DATA_BLOCK "DB %%TAG%%"
{ S7_Optimized_Access := 'FALSE' }
VERSION : 0.1
NON_RETAIN
"@pc FB500 monAI _New"

BEGIN
   SAMPLE_T := 0.1;
   HMI_SIM := TRUE;
   "enAlm AH" := TRUE;
   "enAlm WH" := TRUE;
   "enAlm WL" := TRUE;
   "enAlm AL" := TRUE;
   "enAlm CSF" := TRUE;
   "enAction AH" := TRUE;
   "enAction WH" := TRUE;
   "enAction WL" := TRUE;
   "enAction AL" := TRUE;
   "enAction CSF" := TRUE;
   "exist AH" := FALSE;
   "exist WH" := FALSE;
   "exist WL" := FALSE;
   "exist AL" := FALSE;
   "exist CSF" := FALSE;
   "enCalc AH" := TRUE;
   "enCalc WH" := TRUE;
   "enCalc WL" := TRUE;
   "enCalc AL" := TRUE;
   "enCalc CSF" := TRUE;
   hmiContrBYP := FALSE;
   AH_isTRIP := TRUE;
   WH_isTRIP := FALSE;
   WL_isTRIP := FALSE;
   AL_isTRIP := TRUE;
   CSF_isTRIP := TRUE;
   enSUBS := FALSE;
   pvSUBS := 0.0;
   inDIR := FALSE;
   pvDIR := 0.0;
   inDIR_upLim := 400.0;
   inDIR_loLim := -200.0;
   inChannel := 0;
   inCARD_upLim := 20.0;
   inCARD_loLim := 4.0;
   inRAW_upLim := 27648.0;
   inRAW_loLim := 0.0;
   NM_upLim := 400.0;
   NM_loLim := -200.0;
   CSF_External := FALSE;
   CSF_UpLim := 30000.0;
   CSF_loLim := -30000.0;
   HYS := 0.0;
   timSET_AHOn := 0.0;
   timSET_AHOff := 2.0;
   timSET_WHOn := 0.0;
   timSET_WHOff := 2.0;
   timSET_WLOn := 0.0;
   timSET_WLOff := 2.0;
   timSET_ALOn := 0.0;
   timSET_ALOff := 2.0;
   timSET_CSFOn := 0.0;
   timSET_CSFOff := 2.0;
   qPV := 0.0;
   qmeasPV := 0.0;
   qCARD := 0.0;
   "qAlm AH" := FALSE;
   "qAlm WH" := FALSE;
   "qAlm WL" := FALSE;
   "qAlm AL" := FALSE;
   "qAlm CSF" := FALSE;
   "qAction AH" := FALSE;
   "qAction WH" := FALSE;
   "qAction WL" := FALSE;
   "qAction AL" := FALSE;
   "qAction CSF" := FALSE;
   qContrBYP := FALSE;
   qThrBYP := FALSE;
   qSIM := FALSE;
   qCHF_HL := FALSE;
   qCHF_LL := FALSE;
   qSUBS := FALSE;
   wHMIST := 16#0000;
   wALM := 16#0000;
   U_AH := 100.0;
   U_WH := 100.0;
   U_WL := 0.0;
   U_AL := 0.0;
   pvSIM := 0.0;
   RESET_HMI := FALSE;
   RESET_EVAL := FALSE;
   CSF_DLY_ON := FALSE;
   CSF_DLY_OFF := TRUE;
   AH_DLY_ON := FALSE;
   AH_DLY_OFF := TRUE;
   WH_DLY_ON := FALSE;
   WH_DLY_OFF := FALSE;
   WL_DLY_ON := FALSE;
   WL_DLY_OFF := FALSE;
   AL_DLY_ON := FALSE;
   AL_DLY_OFF := FALSE;
   CSF_GEN := FALSE;
   AH_GEN := FALSE;
   WH_GEN := FALSE;
   WL_GEN := FALSE;
   AL_GEN := FALSE;
   AH_ACT := FALSE;
   WH_ACT := FALSE;
   WL_ACT := FALSE;
   AL_ACT := FALSE;
   CSF_ACT := FALSE;
   MEM_U_IN := 0.0;
   MEM_PV := 0.0;
   Card_UR_DELTA := 16.0;
   MEM_CardPV := 0.0;
   U_HYS := 0.0;
   TIME_CSF_ON := 0.0;
   TIME_CSF_OFF := 2.0;
   TIME_AH_ON := 0.0;
   TIME_AH_OFF := 2.0;
   TIME_WH_ON := 0.0;
   TIME_WH_OFF := 0.0;
   TIME_WL_ON := 0.0;
   TIME_WL_OFF := 0.0;
   TIME_AL_ON := 0.0;
   TIME_AL_OFF := 0.0;
   DESCRIPTION := '%%DESC%%';
   TAG := '%%TAG%%';
   UM := '%%UNIT%%';
   AH_ACT_EXIST := FALSE;
   WH_ACT_EXIST := FALSE;
   WL_ACT_EXIST := FALSE;
   AL_ACT_EXIST := FALSE;
   CSF_ACT_EXIST := FALSE;

END_DATA_BLOCK

